Fanuc KAREL source: XML_ADDTAG.kl

PROGRAM T
%NOLOCKGROUP
VAR
 v0 : FILE
 v1 : STRING[40]
 v2 : INTEGER
 v3 : BOOLEAN
 v4 : INTEGER
 v5 : INTEGER
BEGIN
 XML_ADDTAG(v0, v1, v2, v3, v4, v5)
END T
